// TIA Portal project "T2_BT4_analogCamBienNhiet" (V14)

(* hardware
DEVICE "S7-1200 station_1"  S7-1200 Station
   slot 0: "Rack_0"  S7-1200 Rack  Rack  V1.0
   slot 1: "PLC_1"  CPU 1214C DC/DC/DC  6ES7 214-1AG40-0XB0  V4.2
*)

// ===== PLC "PLC_1"  CPU 1214C DC/DC/DC =====

VAR_GLOBAL   // PLC tag table "Default tag table"
   "stop" AT %I0.0 : Bool;
   "start/stop" AT %I0.2 : Bool;
   "Tag_1" AT %Q0.0 : Bool;
   "Tag_2" AT %IW64 : Int;
   "Tag_3" AT %MD10 : Real;
   "nhiet do thuc te" AT %MD20 : DWord;
   "motor khuay" AT %Q0.1 : Bool;
   "xuoi" AT %Q0.2 : Bool;
   "Tag_4" AT %M0.0 : Bool;
   "nguoc" AT %Q0.3 : Bool;
   "den bao qua nhiet" AT %Q0.4 : Bool;
   "Tag_5" AT %M0.1 : Bool;
   "reset" AT %M0.2 : Bool;
   "ngat" AT %M0.3 : Bool;
END_VAR

// folder: System blocks/Program resources

DATA_BLOCK "IEC_Timer_0_DB"   // DB1
{ S7_Optimized_Access := 'TRUE' }
AUTHOR : Simatic
FAMILY : IEC
NAME : IEC_TMR
VERSION : 1.0
// stored: InstanceOfName IEC_TIMER
"IEC_TIMER"
BEGIN
END_DATA_BLOCK

DATA_BLOCK "IEC_Timer_0_DB_1"   // DB2
{ S7_Optimized_Access := 'TRUE' }
AUTHOR : Simatic
FAMILY : IEC
NAME : IEC_TMR
VERSION : 1.0
// stored: InstanceOfName IEC_TIMER
"IEC_TIMER"
BEGIN
END_DATA_BLOCK

// folder: (top level)

ORGANIZATION_BLOCK "Main"   // OB1, LAD, ProgramCycle
TITLE = "Main Program Sweep (Cycle)"
{ S7_Optimized_Access := 'TRUE' }
VERSION : 0.1
   VAR_INPUT
      Initial_Call : Bool;   // Initial call of this OB
      Remanence : Bool;   // =True, if remanent data are available
   END_VAR
BEGIN

REGION Network 1
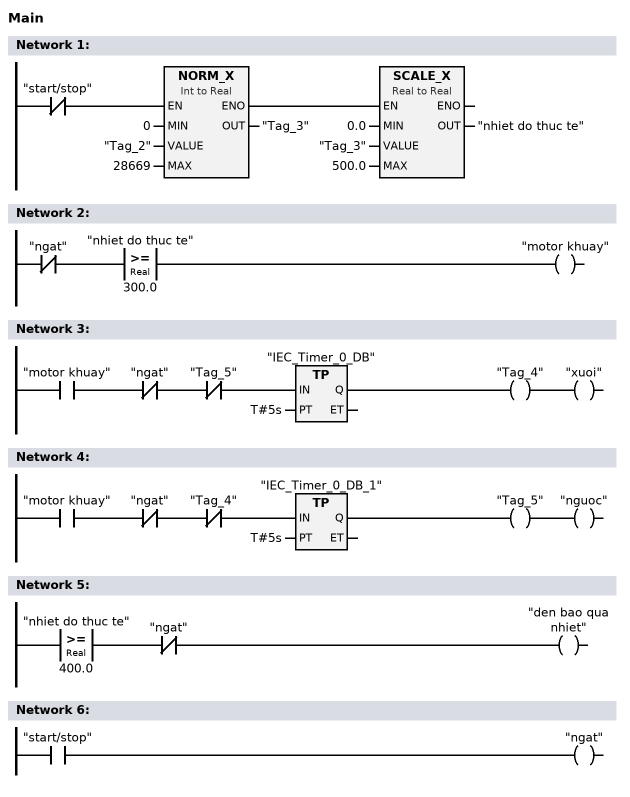
   RUNG wire#powerrail
      I_Contact( "start/stop" )
      { S7_Templates := "[SrcType := Int, DestType := Real]" } Normalize(min := 0, value := "Tag_2", max := 28669, out => "Tag_3")
      { S7_Templates := "[SrcType := Real, DestType := Real]" } Scale(min := 0.0, value := "Tag_3", max := 500.0, out => "nhiet do thuc te")
   END_RUNG
   // the same network as SCL:
   IF NOT "start/stop" THEN
       "Tag_3" := NORM_X(MIN := 0, VALUE := "Tag_2", MAX := 28669);
       "nhiet do thuc te" := SCALE_X(MIN := 0.0, VALUE := "Tag_3", MAX := 500.0);
   END_IF;
END_REGION

REGION Network 2
   RUNG wire#powerrail
      I_Contact( "ngat" )
      { S7_Templates := "SrcType := Real" } GE_Contact(in1 := "nhiet do thuc te", in2 := 300.0)
      Coil( "motor khuay" )
   END_RUNG
   // the same network as SCL:
   "motor khuay" := NOT "ngat" AND ("nhiet do thuc te" >= 300.0);
END_REGION

REGION Network 3
   "IEC_Timer_0_DB".TP(IN := "motor khuay" AND NOT "ngat" AND NOT "Tag_5", PT := T#5s);
   "Tag_4" := "IEC_Timer_0_DB".Q;
   "xuoi" := "IEC_Timer_0_DB".Q;
END_REGION

REGION Network 4
   "IEC_Timer_0_DB_1".TP(IN := "motor khuay" AND NOT "ngat" AND NOT "Tag_4", PT := T#5s);
   "Tag_5" := "IEC_Timer_0_DB_1".Q;
   "nguoc" := "IEC_Timer_0_DB_1".Q;
END_REGION

REGION Network 5
   RUNG wire#powerrail
      { S7_Templates := "SrcType := Real" } GE_Contact(in1 := "nhiet do thuc te", in2 := 400.0)
      I_Contact( "ngat" )
      Coil( "den bao qua nhiet" )
   END_RUNG
   // the same network as SCL:
   "den bao qua nhiet" := ("nhiet do thuc te" >= 400.0) AND NOT "ngat";
END_REGION

REGION Network 6
   RUNG wire#powerrail
      Contact( "start/stop" )
      Coil( "ngat" )
   END_RUNG
   // the same network as SCL:
   "ngat" := "start/stop";
END_REGION
END_ORGANIZATION_BLOCK